# B&R Automation Studio project Teknologia25 (part 10)

#### rotationProgram.st
```iecst
ACTION rotationTask:
	positionContainerRotation[0].initXPos := 0.180;
	positionContainerRotation[0].initYPos := 0.060;
	positionContainerRotation[1].initXPos := 0.060;
	positionContainerRotation[1].initYPos := 0.060;
	positionContainerRotation[2].initXPos := 0.060;
	positionContainerRotation[2].initYPos := 0.180;
	positionContainerRotation[3].initXPos := 0.180;
	positionContainerRotation[3].initYPos := 0.180;

	gWorkStations[0].par.xLocation										:= 0.180;
	gWorkStations[0].par.yLocation										:= 0.060;
	gWorkStations[0].par.nextStationSelector							:= '1';
	gWorkStations[0].par.processTime									:= 0;
	gWorkStations[0].par.pathRouting									:= 1;
	gWorkStations[0].par.landBeforeProcess								:= FALSE;
	gWorkStations[0].par.ArcMovement									:= FALSE;

	gWorkStations[1].par.xLocation										:= 0.060;
	gWorkStations[1].par.yLocation										:= 0.180;
	gWorkStations[1].par.nextStationSelector							:= '0';
	gWorkStations[1].par.processTime									:= WorkStation2And3MovementTimer;
	gWorkStations[1].par.pathRouting									:= 2;
	gWorkStations[1].par.landBeforeProcess								:= TRUE;
	gWorkStations[1].par.ArcMovement									:= FALSE;

	CASE em.substate OF
		14000:
			em.description := 'Move shuttle to pre pos';
			tempShuttleCounter := 0;
			MC_BR_MoveInPlaneAsync_Acp6D_0.Parameters.Acceleration := gAcp6DCtrl.Par.Acceleration;
			MC_BR_MoveInPlaneAsync_Acp6D_0.Parameters.Velocity := gAcp6DCtrl.Par.Velocity;
			FOR i := 0 TO UINT_TO_USINT(localCurrentNumShuttles-1) DO
				MC_BR_MoveInPlaneAsync_Acp6D_0.Parameters.AsyncPar[i].Shuttle := ADR(gAcp6DCtrl.Status.ShuttleInfo[i].shuttleRef);
				MC_BR_MoveInPlaneAsync_Acp6D_0.Parameters.AsyncPar[i].X := positionContainerRotation[i].initXPos;
				MC_BR_MoveInPlaneAsync_Acp6D_0.Parameters.AsyncPar[i].Y := positionContainerRotation[i].initYPos;
			END_FOR
			MC_BR_MoveInPlaneAsync_Acp6D_0.Execute := TRUE;
			IF MC_BR_MoveInPlaneAsync_Acp6D_0.Acknowledge THEN
				MC_BR_MoveInPlaneAsync_Acp6D_0.Execute := FALSE;
				em.substate := 14010;
			END_IF

		14010:
			em.description := 'Move shuttle 2 towards workstation 0';
			MC_BR_MoveInPlane_Acp6D_0.Parameters.Acceleration := gAcp6DCtrl.Par.Acceleration;
			MC_BR_MoveInPlane_Acp6D_0.Parameters.Velocity := gAcp6DCtrl.Par.Velocity;
			MC_BR_MoveInPlane_Acp6D_0.Shuttle := ADR(gAcp6DCtrl.Status.ShuttleInfo[1].shuttleRef);;
			MC_BR_MoveInPlane_Acp6D_0.Parameters.Position.X := gWorkStations[0].par.xLocation;;
			MC_BR_MoveInPlane_Acp6D_0.Parameters.Position.Y := gWorkStations[0].par.yLocation;
			MC_BR_MoveInPlane_Acp6D_0.Parameters.Path := 0; //direct
			MC_BR_MoveInPlane_Acp6D_0.Parameters.Mode := 0;
			MC_BR_MoveInPlane_Acp6D_0.Execute := TRUE;
			IF MC_BR_MoveInPlane_Acp6D_0.Acknowledge THEN
				MC_BR_MoveInPlane_Acp6D_0.Execute := FALSE;
				em.substate := 14020;
			END_IF

		14020:
			em.description := 'Move shuttle 3 towards workstation 0';
			MC_BR_MoveInPlane_Acp6D_0.Parameters.Acceleration := gAcp6DCtrl.Par.Acceleration;
			MC_BR_MoveInPlane_Acp6D_0.Parameters.Velocity := gAcp6DCtrl.Par.Velocity;
			MC_BR_MoveInPlane_Acp6D_0.Shuttle := ADR(gAcp6DCtrl.Status.ShuttleInfo[2].shuttleRef);;
			MC_BR_MoveInPlane_Acp6D_0.Parameters.Position.X := gWorkStations[0].par.xLocation;;
			MC_BR_MoveInPlane_Acp6D_0.Parameters.Position.Y := gWorkStations[0].par.yLocation;
			MC_BR_MoveInPlane_Acp6D_0.Parameters.Path := 2; //Y then X
			MC_BR_MoveInPlane_Acp6D_0.Parameters.Mode := 0;
			MC_BR_MoveInPlane_Acp6D_0.Execute := TRUE;
			IF MC_BR_MoveInPlane_Acp6D_0.Acknowledge THEN
				MC_BR_MoveInPlane_Acp6D_0.Execute := FALSE;
				em.substate := 14030;
			END_IF

		14030:
			em.description := 'Move shuttle 4 towards workstation 1';
			MC_BR_MoveInPlane_Acp6D_0.Parameters.Acceleration := gAcp6DCtrl.Par.Acceleration;
			MC_BR_MoveInPlane_Acp6D_0.Parameters.Velocity := gAcp6DCtrl.Par.Velocity;
			MC_BR_MoveInPlane_Acp6D_0.Shuttle := ADR(gAcp6DCtrl.Status.ShuttleInfo[3].shuttleRef);;
			MC_BR_MoveInPlane_Acp6D_0.Parameters.Position.X := 0.060;
			MC_BR_MoveInPlane_Acp6D_0.Parameters.Position.Y := 0.180;
			MC_BR_MoveInPlane_Acp6D_0.Parameters.Path := 0; //direct
			MC_BR_MoveInPlane_Acp6D_0.Parameters.Mode := 0;
			MC_BR_MoveInPlane_Acp6D_0.Execute := TRUE;
			IF MC_BR_MoveInPlane_Acp6D_0.Acknowledge THEN
				MC_BR_MoveInPlane_Acp6D_0.Execute := FALSE;
				em.substate := 14040;
			END_IF

		14040:
			em.description := 'Move shuttle 4 towards workstation 1';
			MC_BR_MoveInPlane_Acp6D_0.Parameters.Acceleration := gAcp6DCtrl.Par.Acceleration;
			MC_BR_MoveInPlane_Acp6D_0.Parameters.Velocity := gAcp6DCtrl.Par.Velocity;
			MC_BR_MoveInPlane_Acp6D_0.Shuttle := ADR(gAcp6DCtrl.Status.ShuttleInfo[3].shuttleRef);;
			MC_BR_MoveInPlane_Acp6D_0.Parameters.Position.X := gWorkStations[0].par.xLocation;
			MC_BR_MoveInPlane_Acp6D_0.Parameters.Position.Y := gWorkStations[0].par.yLocation;
			MC_BR_MoveInPlane_Acp6D_0.Parameters.Path := 2; //direct
			MC_BR_MoveInPlane_Acp6D_0.Parameters.Mode := 0;
			MC_BR_MoveInPlane_Acp6D_0.Execute := TRUE;
			IF MC_BR_MoveInPlane_Acp6D_0.Acknowledge THEN
				MC_BR_MoveInPlane_Acp6D_0.Execute := FALSE;
				em.substate := 14050;
			END_IF
	END_CASE

END_ACTION

ACTION rotationStation:
	CASE cm.state OF
		// Display station at image
		//'<foreignObject x="20" y="20" width="300" height="300"><img src="Media/statusGreen.png" height="300" width="300"/>'
		//brsstrcat(ADR(showWorkStations),ADR('<foreingObject x="'));
		//brdkStrCat(ADR(showWorkStations), ADR(testDraw));
		//brdkStrCat(ADR(showWorkStations),'<foreingObject x="');

		0:
			//Check what shuttle is on top of workstation
			FOR k := 0 TO NUM_SHUTTLES DO
				IF((gAcp6DCtrl.Status.ShuttleInfo[k].Position.X > pWorkStations.par.xLocation - MARGIN AND gAcp6DCtrl.Status.ShuttleInfo[k].Position.X < pWorkStations.par.xLocation + MARGIN) AND
					gAcp6DCtrl.Status.ShuttleInfo[k].Position.Y > pWorkStations.par.yLocation - MARGIN AND gAcp6DCtrl.Status.ShuttleInfo[k].Position.Y < pWorkStations.par.yLocation + MARGIN) THEN
					IF gAcp6DCtrl.Status.ShuttleInfo[k].State = mcACP6D_SH_STATE_IDLING THEN
						pWorkStations.par.tempShuttleID := k;
						cm.state := 10;
					END_IF
				END_IF
			END_FOR

		10:
			//Move first workstation
			pWorkStations.MC_BR_MoveInPlane_Acp6D_0.Shuttle := ADR(gAcp6DCtrl.Status.ShuttleInfo[pWorkStations.par.tempShuttleID].shuttleRef);
			pWorkStations.MC_BR_MoveInPlane_Acp6D_0.Parameters.Velocity := gAcp6DCtrl.Par.Velocity;
			pWorkStations.MC_BR_MoveInPlane_Acp6D_0.Parameters.Acceleration := gAcp6DCtrl.Par.Acceleration;
			pWorkStations.MC_BR_MoveInPlane_Acp6D_0.Parameters.Position.X := 0.360;
			pWorkStations.MC_BR_MoveInPlane_Acp6D_0.Parameters.Position.Y := 0.120;
			pWorkStations.MC_BR_MoveInPlane_Acp6D_0.Parameters.Mode := 0; //Absolute
			pWorkStations.MC_BR_MoveInPlane_Acp6D_0.Parameters.Path := 1; //0 Diagonal, 1 First X then Y, 2 First Y then X
			pWorkStations.MC_BR_MoveInPlane_Acp6D_0.Execute := TRUE;
			IF pWorkStations.MC_BR_MoveInPlane_Acp6D_0.Done THEN
				pWorkStations.MC_BR_MoveInPlane_Acp6D_0.Execute := FALSE;
				cm.state := 20;
			END_IF

		20:
			//Rotate 90 degress
			em.cmd.sc := FALSE;
			pWorkStations.MC_BR_RotaryMotion_Acp6D_0.Shuttle := ADR(gAcp6DCtrl.Status.ShuttleInfo[pWorkStations.par.tempShuttleID].shuttleRef);
			pWorkStations.MC_BR_RotaryMotion_Acp6D_0.Parameters.Acceleration := gAcp6DCtrl.Par.rotationAcceleration;
			pWorkStations.MC_BR_RotaryMotion_Acp6D_0.Parameters.Velocity := gAcp6DCtrl.Par.rotationVelocity;
			pWorkStations.MC_BR_RotaryMotion_Acp6D_0.Parameters.Angle := 1.57079633; //90 degress
			pWorkStations.MC_BR_RotaryMotion_Acp6D_0.Parameters.Mode := 0;
			pWorkStations.MC_BR_RotaryMotion_Acp6D_0.Execute := TRUE;
			IF pWorkStations.MC_BR_RotaryMotion_Acp6D_0.Done THEN
				pWorkStations.MC_BR_RotaryMotion_Acp6D_0.Execute := FALSE;
				cm.state := 30;
			END_IF

		30:
			//Move
			//em.cmd.sc := FALSE;
			pWorkStations.MC_BR_MoveInPlane_Acp6D_0.Shuttle := ADR(gAcp6DCtrl.Status.ShuttleInfo[pWorkStations.par.tempShuttleID].shuttleRef);
			pWorkStations.MC_BR_MoveInPlane_Acp6D_0.Parameters.Velocity := gAcp6DCtrl.Par.Velocity;
			pWorkStations.MC_BR_MoveInPlane_Acp6D_0.Parameters.Acceleration := gAcp6DCtrl.Par.Acceleration;
			pWorkStations.MC_BR_MoveInPlane_Acp6D_0.Parameters.Position.X := 0.420;
			pWorkStations.MC_BR_MoveInPlane_Acp6D_0.Parameters.Position.Y := 0.120;
			pWorkStations.MC_BR_MoveInPlane_Acp6D_0.Parameters.Mode := 0; //Absolute
			pWorkStations.MC_BR_MoveInPlane_Acp6D_0.Parameters.Path := 1; //0 Diagonal, 1 First X then Y, 2 First Y then X
			pWorkStations.MC_BR_MoveInPlane_Acp6D_0.Execute := TRUE;
			IF pWorkStations.MC_BR_MoveInPlane_Acp6D_0.Acknowledge THEN
				pWorkStations.MC_BR_MoveInPlane_Acp6D_0.Execute := FALSE;
				cm.state := 40;
			END_IF

		40:
			//em.cmd.sc := FALSE;
			pWorkStations.TON_0.IN := TRUE;
			pWorkStations.TON_0.PT := t#100ms;
			IF pWorkStations.TON_0.Q THEN
				pWorkStations.TON_0.IN := FALSE;
				cm.state := 50;
			END_IF

		50:
			//Move
			//em.cmd.sc := FALSE;
			pWorkStations.MC_BR_MoveInPlane_Acp6D_0.Shuttle := ADR(gAcp6DCtrl.Status.ShuttleInfo[pWorkStations.par.tempShuttleID].shuttleRef);
			pWorkStations.MC_BR_MoveInPlane_Acp6D_0.Parameters.Velocity := gAcp6DCtrl.Par.Velocity;
			pWorkStations.MC_BR_MoveInPlane_Acp6D_0.Parameters.Acceleration := gAcp6DCtrl.Par.Acceleration;
			pWorkStations.MC_BR_MoveInPlane_Acp6D_0.Parameters.Position.X := 0.360;
			pWorkStations.MC_BR_MoveInPlane_Acp6D_0.Parameters.Position.Y := 0.120;
			pWorkStations.MC_BR_MoveInPlane_Acp6D_0.Parameters.Mode := 0; //Absolute
			pWorkStations.MC_BR_MoveInPlane_Acp6D_0.Parameters.Path := 1; //0 Diagonal, 1 First X then Y, 2 First Y then X
			pWorkStations.MC_BR_MoveInPlane_Acp6D_0.Execute := TRUE;
			IF pWorkStations.MC_BR_MoveInPlane_Acp6D_0.Acknowledge THEN
				pWorkStations.MC_BR_MoveInPlane_Acp6D_0.Execute := FALSE;
				cm.state := 60;
			END_IF

		60:
			//Rotate 90 degress
			em.cmd.sc := FALSE;
			pWorkStations.MC_BR_RotaryMotion_Acp6D_0.Shuttle := ADR(gAcp6DCtrl.Status.ShuttleInfo[pWorkStations.par.tempShuttleID].shuttleRef);
			pWorkStations.MC_BR_RotaryMotion_Acp6D_0.Parameters.Acceleration := gAcp6DCtrl.Par.rotationAcceleration;
			pWorkStations.MC_BR_RotaryMotion_Acp6D_0.Parameters.Velocity := gAcp6DCtrl.Par.rotationVelocity;
			pWorkStations.MC_BR_RotaryMotion_Acp6D_0.Parameters.Angle := 3.14159265; //180 degress
			pWorkStations.MC_BR_RotaryMotion_Acp6D_0.Parameters.Mode := 0;
			pWorkStations.MC_BR_RotaryMotion_Acp6D_0.Execute := TRUE;
			IF pWorkStations.MC_BR_RotaryMotion_Acp6D_0.Done THEN
				pWorkStations.MC_BR_RotaryMotion_Acp6D_0.Execute := FALSE;
				cm.state := 70;
			END_IF

		70:
			//Move
			//em.cmd.sc := FALSE;
			pWorkStations.MC_BR_MoveInPlane_Acp6D_0.Shuttle := ADR(gAcp6DCtrl.Status.ShuttleInfo[pWorkStations.par.tempShuttleID].shuttleRef);
			pWorkStations.MC_BR_MoveInPlane_Acp6D_0.Parameters.Velocity := gAcp6DCtrl.Par.Velocity;
			pWorkStations.MC_BR_MoveInPlane_Acp6D_0.Parameters.Acceleration := gAcp6DCtrl.Par.Acceleration;
			pWorkStations.MC_BR_MoveInPlane_Acp6D_0.Parameters.Position.X := 0.420;
			pWorkStations.MC_BR_MoveInPlane_Acp6D_0.Parameters.Position.Y := 0.120;
			pWorkStations.MC_BR_MoveInPlane_Acp6D_0.Parameters.Mode := 0; //Absolute
			pWorkStations.MC_BR_MoveInPlane_Acp6D_0.Parameters.Path := 1; //0 Diagonal, 1 First X then Y, 2 First Y then X
			pWorkStations.MC_BR_MoveInPlane_Acp6D_0.Execute := TRUE;
			IF pWorkStations.MC_BR_MoveInPlane_Acp6D_0.Acknowledge THEN
				pWorkStations.MC_BR_MoveInPlane_Acp6D_0.Execute := FALSE;
				cm.state := 80;
			END_IF

		80:
			//em.cmd.sc := FALSE;
			pWorkStations.TON_0.IN := TRUE;
			pWorkStations.TON_0.PT := t#100ms;
			IF pWorkStations.TON_0.Q THEN
				pWorkStations.TON_0.IN := FALSE;
				cm.state := 90;
			END_IF

		90:
			//Move
			//em.cmd.sc := FALSE;
			pWorkStations.MC_BR_MoveInPlane_Acp6D_0.Shuttle := ADR(gAcp6DCtrl.Status.ShuttleInfo[pWorkStations.par.tempShuttleID].shuttleRef);
			pWorkStations.MC_BR_MoveInPlane_Acp6D_0.Parameters.Velocity := gAcp6DCtrl.Par.Velocity;
			pWorkStations.MC_BR_MoveInPlane_Acp6D_0.Parameters.Acceleration := gAcp6DCtrl.Par.Acceleration;
			pWorkStations.MC_BR_MoveInPlane_Acp6D_0.Parameters.Position.X := 0.360;
			pWorkStations.MC_BR_MoveInPlane_Acp6D_0.Parameters.Position.Y := 0.120;
			pWorkStations.MC_BR_MoveInPlane_Acp6D_0.Parameters.Mode := 0; //Absolute
			pWorkStations.MC_BR_MoveInPlane_Acp6D_0.Parameters.Path := 1; //0 Diagonal, 1 First X then Y, 2 First Y then X
			pWorkStations.MC_BR_MoveInPlane_Acp6D_0.Execute := TRUE;
			IF pWorkStations.MC_BR_MoveInPlane_Acp6D_0.Acknowledge THEN
				pWorkStations.MC_BR_MoveInPlane_Acp6D_0.Execute := FALSE;
				cm.state := 100;
			END_IF

		100:
			//Rotate 90 degress
			em.cmd.sc := FALSE;
			pWorkStations.MC_BR_RotaryMotion_Acp6D_0.Shuttle := ADR(gAcp6DCtrl.Status.ShuttleInfo[pWorkStations.par.tempShuttleID].shuttleRef);
			pWorkStations.MC_BR_RotaryMotion_Acp6D_0.Parameters.Acceleration := gAcp6DCtrl.Par.rotationAcceleration;
			pWorkStations.MC_BR_RotaryMotion_Acp6D_0.Parameters.Velocity := gAcp6DCtrl.Par.rotationVelocity;
			pWorkStations.MC_BR_RotaryMotion_Acp6D_0.Parameters.Angle := 4.71238898; //270 degress
			pWorkStations.MC_BR_RotaryMotion_Acp6D_0.Parameters.Mode := 0;
			pWorkStations.MC_BR_RotaryMotion_Acp6D_0.Execute := TRUE;
			IF pWorkStations.MC_BR_RotaryMotion_Acp6D_0.Done THEN
				pWorkStations.MC_BR_RotaryMotion_Acp6D_0.Execute := FALSE;
				cm.state := 110;
			END_IF

		110:
			//Move
			//em.cmd.sc := FALSE;
			pWorkStations.MC_BR_MoveInPlane_Acp6D_0.Shuttle := ADR(gAcp6DCtrl.Status.ShuttleInfo[pWorkStations.par.tempShuttleID].shuttleRef);
			pWorkStations.MC_BR_MoveInPlane_Acp6D_0.Parameters.Velocity := gAcp6DCtrl.Par.Velocity;
			pWorkStations.MC_BR_MoveInPlane_Acp6D_0.Parameters.Acceleration := gAcp6DCtrl.Par.Acceleration;
			pWorkStations.MC_BR_MoveInPlane_Acp6D_0.Parameters.Position.X := 0.420;
			pWorkStations.MC_BR_MoveInPlane_Acp6D_0.Parameters.Position.Y := 0.120;
			pWorkStations.MC_BR_MoveInPlane_Acp6D_0.Parameters.Mode := 0; //Absolute
			pWorkStations.MC_BR_MoveInPlane_Acp6D_0.Parameters.Path := 1; //0 Diagonal, 1 First X then Y, 2 First Y then X
			pWorkStations.MC_BR_MoveInPlane_Acp6D_0.Execute := TRUE;
			IF pWorkStations.MC_BR_MoveInPlane_Acp6D_0.Acknowledge THEN
				pWorkStations.MC_BR_MoveInPlane_Acp6D_0.Execute := FALSE;
				cm.state := 120;
			END_IF

		120:
			//em.cmd.sc := FALSE;
			pWorkStations.TON_0.IN := TRUE;
			pWorkStations.TON_0.PT := t#100ms;
			IF pWorkStations.TON_0.Q THEN
				pWorkStations.TON_0.IN := FALSE;
				cm.state := 130;
			END_IF

		130:
			//Move
			//em.cmd.sc := FALSE;
			pWorkStations.MC_BR_MoveInPlane_Acp6D_0.Shuttle := ADR(gAcp6DCtrl.Status.ShuttleInfo[pWorkStations.par.tempShuttleID].shuttleRef);
			pWorkStations.MC_BR_MoveInPlane_Acp6D_0.Parameters.Velocity := gAcp6DCtrl.Par.Velocity;
			pWorkStations.MC_BR_MoveInPlane_Acp6D_0.Parameters.Acceleration := gAcp6DCtrl.Par.Acceleration;
			pWorkStations.MC_BR_MoveInPlane_Acp6D_0.Parameters.Position.X := 0.360;
			pWorkStations.MC_BR_MoveInPlane_Acp6D_0.Parameters.Position.Y := 0.120;
			pWorkStations.MC_BR_MoveInPlane_Acp6D_0.Parameters.Mode := 0; //Absolute
			pWorkStations.MC_BR_MoveInPlane_Acp6D_0.Parameters.Path := 1; //0 Diagonal, 1 First X then Y, 2 First Y then X
			pWorkStations.MC_BR_MoveInPlane_Acp6D_0.Execute := TRUE;
			IF pWorkStations.MC_BR_MoveInPlane_Acp6D_0.Acknowledge THEN
				pWorkStations.MC_BR_MoveInPlane_Acp6D_0.Execute := FALSE;
				cm.state := 140;
			END_IF

		140:
			//Rotate
			em.cmd.sc := FALSE;
			pWorkStations.MC_BR_RotaryMotion_Acp6D_0.Shuttle := ADR(gAcp6DCtrl.Status.ShuttleInfo[pWorkStations.par.tempShuttleID].shuttleRef);
			pWorkStations.MC_BR_RotaryMotion_Acp6D_0.Parameters.Acceleration := gAcp6DCtrl.Par.rotationAcceleration;
			pWorkStations.MC_BR_RotaryMotion_Acp6D_0.Parameters.Velocity := gAcp6DCtrl.Par.rotationVelocity; //RPM
			pWorkStations.MC_BR_RotaryMotion_Acp6D_0.Parameters.Angle := 0; //0 degress
			pWorkStations.MC_BR_RotaryMotion_Acp6D_0.Parameters.Mode := 1;
			pWorkStations.MC_BR_RotaryMotion_Acp6D_0.Execute := TRUE;
			IF pWorkStations.MC_BR_RotaryMotion_Acp6D_0.Done THEN
				pWorkStations.MC_BR_RotaryMotion_Acp6D_0.Execute := FALSE;
				cm.state := 145;
			END_IF

		145:
			em.cmd.sc := FALSE;
			pWorkStations.MC_BR_RotaryMotionSpin_Acp6D_0.Shuttle := ADR(gAcp6DCtrl.Status.ShuttleInfo[pWorkStations.par.tempShuttleID].shuttleRef);
			pWorkStations.MC_BR_RotaryMotionSpin_Acp6D_0.Parameters.Velocity := gAcp6DCtrl.Par.rotationVelocity;
			pWorkStations.MC_BR_RotaryMotionSpin_Acp6D_0.Parameters.Acceleration := gAcp6DCtrl.Par.rotationAcceleration;
			pWorkStations.MC_BR_RotaryMotionSpin_Acp6D_0.Parameters.Duration := 5;
			pWorkStations.MC_BR_RotaryMotionSpin_Acp6D_0.Execute := TRUE;
			IF pWorkStations.MC_BR_RotaryMotionSpin_Acp6D_0.Done THEN
				pWorkStations.MC_BR_RotaryMotionSpin_Acp6D_0.Execute := FALSE;
				cm.state := 150;
			END_IF

		150:
			//Move
			pWorkStations.MC_BR_MoveInPlane_Acp6D_0.Shuttle := ADR(gAcp6DCtrl.Status.ShuttleInfo[pWorkStations.par.tempShuttleID].shuttleRef);
			pWorkStations.MC_BR_MoveInPlane_Acp6D_0.Parameters.Velocity := gAcp6DCtrl.Par.Velocity;
			pWorkStations.MC_BR_MoveInPlane_Acp6D_0.Parameters.Acceleration := gAcp6DCtrl.Par.Acceleration;
			pWorkStations.MC_BR_MoveInPlane_Acp6D_0.Parameters.Position.X := 0.060;
			pWorkStations.MC_BR_MoveInPlane_Acp6D_0.Parameters.Position.Y := 0.180;
			pWorkStations.MC_BR_MoveInPlane_Acp6D_0.Parameters.Mode := 0; //Absolute
			pWorkStations.MC_BR_MoveInPlane_Acp6D_0.Parameters.Path := 2; //0 Diagonal, 1 First X then Y, 2 First Y then X
			pWorkStations.MC_BR_MoveInPlane_Acp6D_0.Execute := TRUE;
			IF pWorkStations.MC_BR_MoveInPlane_Acp6D_0.Acknowledge THEN
				pWorkStations.MC_BR_MoveInPlane_Acp6D_0.Execute := FALSE;
				cm.state := 160;
			END_IF

		160:
			//Move
			pWorkStations.MC_BR_MoveInPlane_Acp6D_0.Shuttle := ADR(gAcp6DCtrl.Status.ShuttleInfo[pWorkStations.par.tempShuttleID].shuttleRef);
			pWorkStations.MC_BR_MoveInPlane_Acp6D_0.Parameters.Velocity := gAcp6DCtrl.Par.Velocity;
			pWorkStations.MC_BR_MoveInPlane_Acp6D_0.Parameters.Acceleration := gAcp6DCtrl.Par.Acceleration;
			pWorkStations.MC_BR_MoveInPlane_Acp6D_0.Parameters.Position.X := gWorkStations[0].par.xLocation;
			pWorkStations.MC_BR_MoveInPlane_Acp6D_0.Parameters.Position.Y := gWorkStations[0].par.yLocation;
			pWorkStations.MC_BR_MoveInPlane_Acp6D_0.Parameters.Mode := 0; //Absolute
			pWorkStations.MC_BR_MoveInPlane_Acp6D_0.Parameters.Path := 2; //0 Diagonal, 1 First X then Y, 2 First Y then X
			pWorkStations.MC_BR_MoveInPlane_Acp6D_0.Execute := TRUE;
			IF pWorkStations.MC_BR_MoveInPlane_Acp6D_0.Acknowledge THEN
				pWorkStations.MC_BR_MoveInPlane_Acp6D_0.Execute := FALSE;
				cm.state := 0;
			END_IF

	END_CASE

	//Calls
	pWorkStations.MC_BR_MoveInPlane_Acp6D_0();
	pWorkStations.MC_BR_MoveArc_Acp6D_0();
	pWorkStations.MC_BR_ShLevitation_Acp6D_0();
	pWorkStations.MC_BR_RotaryMotion_Acp6D_0();
	pWorkStations.MC_BR_RotaryMotionSpin_Acp6D_0();
	pWorkStations.TON_0();
	cm();

END_ACTION
```

#### steelSheet.st
```iecst
ACTION steelSheetTask:
	positionContainerSteelSheet[0].initXPos := 0.060;
	positionContainerSteelSheet[0].initYPos := 0.060;
	positionContainerSteelSheet[1].initXPos := 0.180;
	positionContainerSteelSheet[1].initYPos := 0.060;
	positionContainerSteelSheet[2].initXPos := 0.300;
	positionContainerSteelSheet[2].initYPos := 0.060;
	positionContainerSteelSheet[3].initXPos := 0.420;
	positionContainerSteelSheet[3].initYPos := 0.060;

	gWorkStations[0].par.xLocation										:= 0.060;
	gWorkStations[0].par.yLocation										:= 0.060;
	gWorkStations[0].par.nextStationSelector							:= '0';
	gWorkStations[0].par.processTime									:= 0;
	gWorkStations[0].par.pathRouting									:= 0;
	gWorkStations[0].par.landBeforeProcess								:= FALSE;
	gWorkStations[0].par.ArcMovement									:= FALSE;

	gWorkStations[1].par.xLocation										:= 0.180;
	gWorkStations[1].par.yLocation										:= 0.060;
	gWorkStations[1].par.nextStationSelector							:= '1';
	gWorkStations[1].par.processTime									:= 0;
	gWorkStations[1].par.pathRouting									:= 0;
	gWorkStations[1].par.landBeforeProcess								:= FALSE;
	gWorkStations[1].par.ArcMovement									:= FALSE;

	gWorkStations[2].par.xLocation										:= 0.300;
	gWorkStations[2].par.yLocation										:= 0.060;
	gWorkStations[2].par.nextStationSelector							:= '2';
	gWorkStations[2].par.processTime									:= 0;
	gWorkStations[2].par.pathRouting									:= 0;
	gWorkStations[2].par.landBeforeProcess								:= FALSE;
	gWorkStations[2].par.ArcMovement									:= FALSE;

	gWorkStations[3].par.xLocation										:= 0.420;
	gWorkStations[3].par.yLocation										:= 0.060;
	gWorkStations[3].par.nextStationSelector							:= '3';
	gWorkStations[3].par.processTime									:= 0;
	gWorkStations[3].par.pathRouting									:= 0;
	gWorkStations[3].par.landBeforeProcess								:= FALSE;
	gWorkStations[3].par.ArcMovement									:= FALSE;

	// Make sure all shuttles have finish movement
	sheetMoveDone := TRUE;
//	FOR i := 0 TO NR_OF_WORKSTATIONS DO
//		IF NOT gWorkStations[i].MC_BR_Move6D_Acp6D_0.Done THEN
//			sheetMoveDone := FALSE;
//		END_IF
//	END_FOR
	FOR i := 0 TO NR_OF_WORKSTATIONS DO
		IF NOT gWorkStations[i].MC_BR_MoveInPlane_Acp6D_0.Done THEN
			sheetMoveDone := FALSE;
		END_IF
	END_FOR

	CASE em.substate OF
		15000:
			em.description := 'Move shuttle to pre pos';
			tempShuttleCounter := 0;
			MC_BR_MoveInPlaneAsync_Acp6D_0.Parameters.Acceleration := gAcp6DCtrl.Par.Acceleration;
			MC_BR_MoveInPlaneAsync_Acp6D_0.Parameters.Velocity := gAcp6DCtrl.Par.Velocity;
			FOR i := 0 TO UINT_TO_USINT(localCurrentNumShuttles-1) DO
				MC_BR_MoveInPlaneAsync_Acp6D_0.Parameters.AsyncPar[i].Shuttle := ADR(gAcp6DCtrl.Status.ShuttleInfo[i].shuttleRef);
				MC_BR_MoveInPlaneAsync_Acp6D_0.Parameters.AsyncPar[i].X := positionContainerSteelSheet[i].initXPos;
				MC_BR_MoveInPlaneAsync_Acp6D_0.Parameters.AsyncPar[i].Y := positionContainerSteelSheet[i].initYPos;
				MC_BR_MoveInPlaneAsync_Acp6D_0.Parameters.AsyncPar[i].Y := positionContainerSteelSheet[i].initYPos;
			END_FOR
			MC_BR_MoveInPlaneAsync_Acp6D_0.Execute := TRUE;
			IF MC_BR_MoveInPlaneAsync_Acp6D_0.Acknowledge THEN
				MC_BR_MoveInPlaneAsync_Acp6D_0.Execute := FALSE;
				em.substate := 15010;
			END_IF

		15010:
			em.description := 'Shuttle moves at a higher levitation hight';

	END_CASE

END_ACTION

ACTION steelSheetStation:
	CASE cm.state OF
		0:
			//Check what shuttle is on top of workstation
			FOR k := 0 TO NUM_SHUTTLES DO
				IF((gAcp6DCtrl.Status.ShuttleInfo[k].Position.X > pWorkStations.par.xLocation - MARGIN AND gAcp6DCtrl.Status.ShuttleInfo[k].Position.X < pWorkStations.par.xLocation + MARGIN) AND
					gAcp6DCtrl.Status.ShuttleInfo[k].Position.Y > pWorkStations.par.yLocation - MARGIN AND gAcp6DCtrl.Status.ShuttleInfo[k].Position.Y < pWorkStations.par.yLocation + MARGIN) THEN
					IF gAcp6DCtrl.Status.ShuttleInfo[k].State = mcACP6D_SH_STATE_IDLING THEN
						pWorkStations.par.tempShuttleID := k;
						cm.state := 5;
					END_IF
				END_IF
			END_FOR

		5:
			// Levitate to sheet flying height
			pWorkStations.MC_BR_MoveShortAxis_Acp6D_0.Shuttle := ADR(gAcp6DCtrl.Status.ShuttleInfo[pWorkStations.par.tempShuttleID].shuttleRef);
			pWorkStations.MC_BR_MoveShortAxis_Acp6D_0.Parameters.Position.Z := steelSheetFlyingHeight;
			pWorkStations.MC_BR_MoveShortAxis_Acp6D_0.Parameters.Position.Rx := 0;
			pWorkStations.MC_BR_MoveShortAxis_Acp6D_0.Parameters.Position.Ry := 0;
			pWorkStations.MC_BR_MoveShortAxis_Acp6D_0.Parameters.Position.Rz := 0;
			pWorkStations.MC_BR_MoveShortAxis_Acp6D_0.Parameters.Velocity.Z := 0.01;
			pWorkStations.MC_BR_MoveShortAxis_Acp6D_0.Execute := TRUE;
			IF pWorkStations.MC_BR_MoveShortAxis_Acp6D_0.Done THEN
				pWorkStations.MC_BR_MoveShortAxis_Acp6D_0.Execute := FALSE;
				cm.state := 10;
			END_IF

		10:
//			pWorkStations.MC_BR_Move6D_Acp6D_0.Shuttle := ADR(gAcp6DCtrl.Status.ShuttleInfo[pWorkStations.par.tempShuttleID].shuttleRef);
//			pWorkStations.MC_BR_Move6D_Acp6D_0.Parameters.InPlane.Velocity := stainlessVelocity;
//			pWorkStations.MC_BR_Move6D_Acp6D_0.Parameters.InPlane.Acceleration := stainlessAcceleration;
//			pWorkStations.MC_BR_Move6D_Acp6D_0.Parameters.InPlane.Position.X := pWorkStations.par.xLocation;
//			pWorkStations.MC_BR_Move6D_Acp6D_0.Parameters.InPlane.Position.Y := 0.180;
//			pWorkStations.MC_BR_Move6D_Acp6D_0.Parameters.ShortAxis.Position.Z := steelSheetFlyingHeight;
//			pWorkStations.MC_BR_Move6D_Acp6D_0.Parameters.ShortAxis.Position.Rx := 0;
//			pWorkStations.MC_BR_Move6D_Acp6D_0.Parameters.ShortAxis.Position.Ry := 0;
//			pWorkStations.MC_BR_Move6D_Acp6D_0.Parameters.ShortAxis.Position.Rz := 0;
//			pWorkStations.MC_BR_Move6D_Acp6D_0.Execute := TRUE;
//			IF pWorkStations.MC_BR_Move6D_Acp6D_0.Done AND sheetMoveDone THEN
//				pWorkStations.MC_BR_Move6D_Acp6D_0.Execute := FALSE;
//				cm.state := 30;
//			END_IF

			pWorkStations.MC_BR_MoveInPlane_Acp6D_0.Shuttle := ADR(gAcp6DCtrl.Status.ShuttleInfo[pWorkStations.par.tempShuttleID].shuttleRef);
			pWorkStations.MC_BR_MoveInPlane_Acp6D_0.Parameters.Velocity := stainlessVelocity;
			pWorkStations.MC_BR_MoveInPlane_Acp6D_0.Parameters.Acceleration := stainlessAcceleration;
			pWorkStations.MC_BR_MoveInPlane_Acp6D_0.Parameters.Position.X := pWorkStations.par.xLocation;
			pWorkStations.MC_BR_MoveInPlane_Acp6D_0.Parameters.Position.Y := 0.180;

			pWorkStations.MC_BR_MoveInPlane_Acp6D_0.Execute := TRUE;
			IF pWorkStations.MC_BR_MoveInPlane_Acp6D_0.Done AND sheetMoveDone THEN
				pWorkStations.MC_BR_MoveInPlane_Acp6D_0.Execute := FALSE;
				cm.state := 15;
			END_IF

		15:
			pWorkStations.TON_0.IN := TRUE;
			pWorkStations.TON_0.PT := stainlessWaitTime;
			IF pWorkStations.TON_0.Q THEN
				pWorkStations.TON_0.IN := FALSE;
				cm.state := 30;
			END_IF

		30:
//			pWorkStations.MC_BR_Move6D_Acp6D_0.Shuttle := ADR(gAcp6DCtrl.Status.ShuttleInfo[pWorkStations.par.tempShuttleID].shuttleRef);
//			pWorkStations.MC_BR_Move6D_Acp6D_0.Parameters.InPlane.Velocity := stainlessVelocity;
//			pWorkStations.MC_BR_Move6D_Acp6D_0.Parameters.InPlane.Acceleration := stainlessAcceleration;
//			pWorkStations.MC_BR_Move6D_Acp6D_0.Parameters.InPlane.Position.X := pWorkStations.par.xLocation;
//			pWorkStations.MC_BR_Move6D_Acp6D_0.Parameters.InPlane.Position.Y := 0.060;
//			pWorkStations.MC_BR_Move6D_Acp6D_0.Parameters.ShortAxis.Position.Rx := 0;
//			pWorkStations.MC_BR_Move6D_Acp6D_0.Parameters.ShortAxis.Position.Ry := 0;
//			pWorkStations.MC_BR_Move6D_Acp6D_0.Parameters.ShortAxis.Position.Rz := 0;
//			pWorkStations.MC_BR_Move6D_Acp6D_0.Parameters.ShortAxis.Position.Z := steelSheetFlyingHeight;
//			pWorkStations.MC_BR_Move6D_Acp6D_0.Execute := TRUE;
//			IF pWorkStations.MC_BR_Move6D_Acp6D_0.Done AND sheetMoveDone THEN
//				pWorkStations.MC_BR_Move6D_Acp6D_0.Execute := FALSE;
//				cm.state := 0;
//			END_IF

			pWorkStations.MC_BR_MoveInPlane_Acp6D_0.Shuttle := ADR(gAcp6DCtrl.Status.ShuttleInfo[pWorkStations.par.tempShuttleID].shuttleRef);
			pWorkStations.MC_BR_MoveInPlane_Acp6D_0.Parameters.Velocity := stainlessVelocity;
			pWorkStations.MC_BR_MoveInPlane_Acp6D_0.Parameters.Acceleration := stainlessAcceleration;
			pWorkStations.MC_BR_MoveInPlane_Acp6D_0.Parameters.Position.X := pWorkStations.par.xLocation;
			pWorkStations.MC_BR_MoveInPlane_Acp6D_0.Parameters.Position.Y := 0.060;

			pWorkStations.MC_BR_MoveInPlane_Acp6D_0.Execute := TRUE;
			IF pWorkStations.MC_BR_MoveInPlane_Acp6D_0.Done AND sheetMoveDone THEN
				pWorkStations.MC_BR_MoveInPlane_Acp6D_0.Execute := FALSE;
				cm.state := 35;
			END_IF

		35:
			pWorkStations.TON_0.IN := TRUE;
			pWorkStations.TON_0.PT := stainlessWaitTime;
			IF pWorkStations.TON_0.Q THEN
				pWorkStations.TON_0.IN := FALSE;
				cm.state := 10;
			END_IF

	END_CASE

	//Calls
	pWorkStations.MC_BR_MoveInPlane_Acp6D_0();
	pWorkStations.MC_BR_MoveArc_Acp6D_0();
	pWorkStations.MC_BR_Move6D_Acp6D_0();
	pWorkStations.MC_BR_ShLevitation_Acp6D_0();
	pWorkStations.MC_BR_RotaryMotion_Acp6D_0();
	pWorkStations.MC_BR_RotaryMotionSpin_Acp6D_0();
	pWorkStations.MC_BR_MoveShortAxis_Acp6D_0();
	pWorkStations.TON_0();
	cm();

END_ACTION
```

#### teachShuttle.st
```iecst
ACTION teachShuttleProgram:
	//setup
	positionContainerFlaskProgram[0].initXPos := 0.060;
	positionContainerFlaskProgram[0].initYPos := 0.060;
	positionContainerFlaskProgram[1].initXPos := 0.060;
	positionContainerFlaskProgram[1].initYPos := 0.180;
	positionContainerFlaskProgram[2].initXPos := 0.180;
	positionContainerFlaskProgram[2].initYPos := 0.120;
	positionContainerFlaskProgram[3].initXPos := 0.360;
	positionContainerFlaskProgram[3].initYPos := 0.120;
	CASE em.substate OF
		16000:
			em.cmd.sc := FALSE;
			em.description := 'Move shuttle to pre pos';
			tempShuttleCounter := 0;
			MC_BR_MoveInPlaneAsync_Acp6D_0.Parameters.Acceleration := gAcp6DCtrl.Par.Acceleration;
			MC_BR_MoveInPlaneAsync_Acp6D_0.Parameters.Velocity := gAcp6DCtrl.Par.Velocity;
			FOR i := 0 TO UINT_TO_USINT(localCurrentNumShuttles-1) DO
				MC_BR_MoveInPlaneAsync_Acp6D_0.Parameters.AsyncPar[i].Shuttle := ADR(gAcp6DCtrl.Status.ShuttleInfo[i].shuttleRef);
				MC_BR_MoveInPlaneAsync_Acp6D_0.Parameters.AsyncPar[i].X := positionContainerFlaskProgram[i].initXPos;
				MC_BR_MoveInPlaneAsync_Acp6D_0.Parameters.AsyncPar[i].Y := positionContainerFlaskProgram[i].initYPos;
			END_FOR
			MC_BR_MoveInPlaneAsync_Acp6D_0.Execute := TRUE;
			IF MC_BR_MoveInPlaneAsync_Acp6D_0.Done THEN
				MC_BR_MoveInPlaneAsync_Acp6D_0.Execute := FALSE;
				em.substate := 16010;
			END_IF

		16010:
			em.cmd.sc := FALSE;
			em.description := 'Deactivate segment 2';
			MC_BR_SegPowerOff_Acp6D_0.Segment := ADR(gAcp6DCtrl.Status.SegmentInfo[1].segmentRef);
			MC_BR_SegPowerOff_Acp6D_0.Execute := TRUE;
			IF MC_BR_SegPowerOff_Acp6D_0.Done THEN
				shuttleDeativatedLock := TRUE;
				MC_BR_SegPowerOff_Acp6D_0.Execute := FALSE;
				em.substate := 16020;
			END_IF

		16020:
			em.cmd.sc := FALSE;
			em.description := 'Menu';
			IF teachProgram.teachPosCmd THEN
				teachProgram.teachPosCmd := FALSE;
				em.substate := 16100;
			ELSIF teachProgram.runProgram THEN
				teachProgram.runProgram := FALSE;
				teachProgram.tmpRunPosCnt := 0;
				em.substate := 16200;
			ELSIF teachProgram.clearPositions THEN
				FOR i := 0 TO 99 DO
					teachProgram.positionArray[i].xPos := 0;
					teachProgram.positionArray[i].yPos := 0;
					teachProgram.savedPositions := 0;
				END_FOR
			ELSIF gAcp6DCtrl.Par.modeSelector <> teachProgramEnum THEN
				em.substate := 16300;
			END_IF

		16100:
			em.cmd.sc := FALSE;
			em.description := 'Teach Position';
			IF gAcp6DCtrl.Status.ShuttleInfo[3].State = mcACP6D_SH_STATE_DISABLED THEN
				teachProgram.positionArray[teachProgram.savedPositions].xPos := gAcp6DCtrl.Status.ShuttleInfo[3].Position.X;
				teachProgram.positionArray[teachProgram.savedPositions].yPos := gAcp6DCtrl.Status.ShuttleInfo[3].Position.Y;
//				teachProgram.positionArray[teachProgram.savedPositions].zPos := gAcp6DCtrl.Status.ShuttleInfo[3].Position.Z;
//				teachProgram.positionArray[teachProgram.savedPositions].rxPos := gAcp6DCtrl.Status.ShuttleInfo[3].Position.Rx;
//				teachProgram.positionArray[teachProgram.savedPositions].ryPos := gAcp6DCtrl.Status.ShuttleInfo[3].Position.Ry;
//				teachProgram.positionArray[teachProgram.savedPositions].rzPos := gAcp6DCtrl.Status.ShuttleInfo[3].Position.Rz;
				teachProgram.savedPositions := teachProgram.savedPositions + 1;
				em.substate := 16020;
			ELSE
				em.substate := 16020;
			END_IF

		16200:
			em.cmd.sc := FALSE;
			MC_BR_SegPowerOn_Acp6D_0.Segment := ADR(gAcp6DCtrl.Status.SegmentInfo[1].segmentRef);
			MC_BR_SegPowerOn_Acp6D_0.Execute := TRUE;
			IF MC_BR_SegPowerOn_Acp6D_0.Done THEN
				MC_BR_SegPowerOn_Acp6D_0.Execute := FALSE;
				em.substate := 16210;
			END_IF

		16210:
			em.cmd.sc := FALSE;
			em.description := 'Run teached program';
			IF teachProgram.tmpRunPosCnt >= teachProgram.savedPositions THEN
				em.substate := 16230;
			ELSE
				em.substate := 16220;
			END_IF

		16220:
			em.cmd.sc := FALSE;
			em.description := 'Run next position in program';
			MC_BR_Move6D_Acp6D_0.Shuttle := ADR(gAcp6DCtrl.Status.ShuttleInfo[3].shuttleRef);
			MC_BR_Move6D_Acp6D_0.Parameters.InPlane.Position.X := teachProgram.positionArray[teachProgram.tmpRunPosCnt].xPos;
			MC_BR_Move6D_Acp6D_0.Parameters.InPlane.Position.Y := teachProgram.positionArray[teachProgram.tmpRunPosCnt].yPos;
			MC_BR_Move6D_Acp6D_0.Parameters.ShortAxis.Position.Z := 0.001;
			MC_BR_Move6D_Acp6D_0.Parameters.InPlane.Velocity := gAcp6DCtrl.Par.Velocity;
			MC_BR_Move6D_Acp6D_0.Parameters.InPlane.Acceleration := gAcp6DCtrl.Par.Acceleration;
			MC_BR_Move6D_Acp6D_0.Parameters.ShortAxis.Velocity.Rx := 1;
			MC_BR_Move6D_Acp6D_0.Parameters.ShortAxis.Velocity.Ry := 1;
			MC_BR_Move6D_Acp6D_0.Parameters.ShortAxis.Velocity.Rz := 1;
			MC_BR_Move6D_Acp6D_0.Parameters.ShortAxis.Velocity.Z := 1;
			MC_BR_Move6D_Acp6D_0.Parameters.ShortAxis.Position.Rz := teachProgram.positionArray[teachProgram.tmpRunPosCnt].rzPos;
			MC_BR_Move6D_Acp6D_0.Execute := TRUE;
			IF MC_BR_Move6D_Acp6D_0.Done THEN
				MC_BR_Move6D_Acp6D_0.Execute := FALSE;
				teachProgram.tmpRunPosCnt := teachProgram.tmpRunPosCnt + 1;
				em.substate := 16210;
			END_IF

		16230:
			em.cmd.sc := FALSE;
			em.description := 'Turn off segment before reteaching';
			MC_BR_SegPowerOff_Acp6D_0.Segment := ADR(gAcp6DCtrl.Status.SegmentInfo[1].segmentRef);
			MC_BR_SegPowerOff_Acp6D_0.Execute := TRUE;
			IF MC_BR_SegPowerOff_Acp6D_0.Done THEN
				MC_BR_SegPowerOff_Acp6D_0.Execute := FALSE;
				em.substate := 16020;
			END_IF

		16300:
			em.cmd.sc := FALSE;
			em.description := 'Power on segment before program change';
			MC_BR_SegPowerOn_Acp6D_0.Segment := ADR(gAcp6DCtrl.Status.SegmentInfo[1].segmentRef);
			MC_BR_SegPowerOn_Acp6D_0.Execute := TRUE;
			IF MC_BR_SegPowerOn_Acp6D_0.Done THEN
				MC_BR_SegPowerOn_Acp6D_0.Execute := FALSE;
				em.substate := 16310;
			END_IF

		16310:
			em.description := 'Check that shuttle is rdy';
			IF gAcp6DCtrl.Status.ShuttleInfo[3].State = mcACP6D_SH_STATE_IDLING THEN
				MC_BR_SegBarrierCommand_Acp6D_0.Segment := ADR(gAcp6DCtrl.Status.SegmentInfo[1].segmentRef);
				MC_BR_SegBarrierCommand_Acp6D_0.Parameters.Command := mcACP6D_BARRIER_OPEN;
				MC_BR_SegBarrierCommand_Acp6D_0.Execute := TRUE;
				IF MC_BR_SegBarrierCommand_Acp6D_0.Done THEN
					MC_BR_SegBarrierCommand_Acp6D_0.Execute := FALSE;
					shuttleDeativatedLock := FALSE;
					em.cmd.sc := TRUE;
				END_IF
			END_IF

	END_CASE

END_ACTION
```

#### trakMode.st
```iecst
ACTION trakModeTask:

	CASE em.substate OF
		17000:
			em.cmd.sc := FALSE;
			em.description := 'Move shuttle to pre pos';
			positionContainerTrakMode[0].initXPos := 0.060;
			positionContainerTrakMode[0].initYPos := 0.060;
			positionContainerTrakMode[1].initXPos := 0.060;
			positionContainerTrakMode[1].initYPos := 0.180;
			positionContainerTrakMode[2].initXPos := 0.300;
			positionContainerTrakMode[2].initYPos := 0.180;
			positionContainerTrakMode[3].initXPos := 0.420;
			positionContainerTrakMode[3].initYPos := 0.180;
			tempShuttleCounter := 0;
			MC_BR_MoveInPlaneAsync_Acp6D_0.Parameters.Acceleration := gAcp6DCtrl.Par.Acceleration;
			MC_BR_MoveInPlaneAsync_Acp6D_0.Parameters.Velocity := gAcp6DCtrl.Par.Velocity;
			FOR i := 0 TO UINT_TO_USINT(localCurrentNumShuttles-1) DO
				MC_BR_MoveInPlaneAsync_Acp6D_0.Parameters.AsyncPar[i].Shuttle := ADR(gAcp6DCtrl.Status.ShuttleInfo[i].shuttleRef);
				MC_BR_MoveInPlaneAsync_Acp6D_0.Parameters.AsyncPar[i].X := positionContainerTrakMode[i].initXPos;
				MC_BR_MoveInPlaneAsync_Acp6D_0.Parameters.AsyncPar[i].Y := positionContainerTrakMode[i].initYPos;
			END_FOR
			MC_BR_MoveInPlaneAsync_Acp6D_0.Execute := TRUE;
			IF MC_BR_MoveInPlaneAsync_Acp6D_0.Done THEN
				MC_BR_MoveInPlaneAsync_Acp6D_0.Execute := FALSE;
				em.substate := 17010;
			END_IF

		17010:
		//HMI interface
			IF trakMode.bigBottle THEN
				em.substate := 17100;
				trakMode.bigBottle := FALSE;
			ELSIF trakMode.smallBottle THEN
				em.substate := 17200;
				trakMode.smallBottle := FALSE;
			END_IF

		17100:
			em.description := 'adjust shuttle to bigBottle';
			MC_BR_MoveInPlane_Acp6D_0.Shuttle := ADR(gAcp6DCtrl.Status.ShuttleInfo[2].shuttleRef);
			MC_BR_MoveInPlane_Acp6D_0.Parameters.Position.X := 0.276;
			MC_BR_MoveInPlane_Acp6D_0.Parameters.Position.Y := 0.180;
			MC_BR_MoveInPlane_Acp6D_0.Parameters.Velocity := gAcp6DCtrl.Par.Velocity;
			MC_BR_MoveInPlane_Acp6D_0.Parameters.Acceleration := gAcp6DCtrl.Par.Acceleration;
			MC_BR_MoveInPlane_Acp6D_0.Parameters.Mode := 0;
			MC_BR_MoveInPlane_Acp6D_0.Parameters.Path := 0;
			MC_BR_MoveInPlane_Acp6D_0.Execute := TRUE;
			IF MC_BR_MoveInPlane_Acp6D_0.Acknowledge THEN
				MC_BR_MoveInPlane_Acp6D_0.Execute := FALSE;
				em.substate := 17500;
			END_IF

		17200:
			em.description := 'adjust shuttle to smallBottle';
			MC_BR_MoveInPlane_Acp6D_0.Shuttle := ADR(gAcp6DCtrl.Status.ShuttleInfo[2].shuttleRef);
			MC_BR_MoveInPlane_Acp6D_0.Parameters.Position.X := 0.293;
			MC_BR_MoveInPlane_Acp6D_0.Parameters.Position.Y := 0.180;
			MC_BR_MoveInPlane_Acp6D_0.Parameters.Velocity := gAcp6DCtrl.Par.Velocity;
			MC_BR_MoveInPlane_Acp6D_0.Parameters.Acceleration := gAcp6DCtrl.Par.Acceleration;
			MC_BR_MoveInPlane_Acp6D_0.Parameters.Mode := 0;
			MC_BR_MoveInPlane_Acp6D_0.Parameters.Path := 0;
			MC_BR_MoveInPlane_Acp6D_0.Execute := TRUE;
			IF MC_BR_MoveInPlane_Acp6D_0.Acknowledge THEN
				MC_BR_MoveInPlane_Acp6D_0.Execute := FALSE;
				em.substate := 17500;
			END_IF

		17500:
			em.description := 'Couple ShuttleGroup3_4';
			em.cmd.sc := FALSE;
			MC_BR_ShGroupCoupleCtrl_Acp6D_0.ShuttleGroup := shGroupShuttle3_4;
			MC_BR_ShGroupCoupleCtrl_Acp6D_0.Parameters.Mode := 1;
			MC_BR_ShGroupCoupleCtrl_Acp6D_0.Parameters.Option := 1; //Couple
			MC_BR_ShGroupCoupleCtrl_Acp6D_0.Execute := TRUE;
			IF MC_BR_ShGroupCoupleCtrl_Acp6D_0.Done THEN
				MC_BR_ShGroupCoupleCtrl_Acp6D_0.Execute := FALSE;
				em.substate := 17550;
			END_IF

		17550:
			em.description := 'Wait timer';
			em.cmd.sc := FALSE;
			TON_0.PT := t#3s;
			TON_0.IN := TRUE;
			IF TON_0.Q THEN
				TON_0.IN := FALSE;
				em.substate := 17600;
			END_IF

		17600:
			em.description := 'Move bottle';
			em.cmd.sc := FALSE;
			MC_BR_MoveInPlane_Acp6D_0.Shuttle := ADR(gAcp6DCtrl.Status.ShuttleInfo[2].shuttleRef);
			MC_BR_MoveInPlane_Acp6D_0.Parameters.Position.X := 0.180;
			MC_BR_MoveInPlane_Acp6D_0.Parameters.Position.Y := 0.180;
			MC_BR_MoveInPlane_Acp6D_0.Parameters.Velocity := 0.5;
			MC_BR_MoveInPlane_Acp6D_0.Parameters.Acceleration := 0.5;
			MC_BR_MoveInPlane_Acp6D_0.Parameters.Mode := 0;
			MC_BR_MoveInPlane_Acp6D_0.Parameters.Path := 0;
			MC_BR_MoveInPlane_Acp6D_0.Execute := TRUE;
			IF MC_BR_MoveInPlane_Acp6D_0.Acknowledge THEN
				MC_BR_MoveInPlane_Acp6D_0.Execute := FALSE;
				em.substate := 17610;
			END_IF

		17610:
			em.description := 'Move bottle';
			em.cmd.sc := FALSE;
			MC_BR_MoveInPlane_Acp6D_0.Shuttle := ADR(gAcp6DCtrl.Status.ShuttleInfo[3].shuttleRef);
			MC_BR_MoveInPlane_Acp6D_0.Parameters.Position.X := 0.420;
			MC_BR_MoveInPlane_Acp6D_0.Parameters.Position.Y := 0.180;
			MC_BR_MoveInPlane_Acp6D_0.Parameters.Velocity := 0.5;
			MC_BR_MoveInPlane_Acp6D_0.Parameters.Acceleration := 0.5;
			MC_BR_MoveInPlane_Acp6D_0.Parameters.Mode := 0;
			MC_BR_MoveInPlane_Acp6D_0.Parameters.Path := 0;
			MC_BR_MoveInPlane_Acp6D_0.Execute := TRUE;
			IF MC_BR_MoveInPlane_Acp6D_0.Acknowledge THEN
				MC_BR_MoveInPlane_Acp6D_0.Execute := FALSE;
				em.substate := 17700;
			END_IF

		17700:
			em.description := 'DeCouple ShuttleGroup3_4';
			em.cmd.sc := FALSE;
			MC_BR_ShGroupCoupleCtrl_Acp6D_0.ShuttleGroup := shGroupShuttle3_4;
			MC_BR_ShGroupCoupleCtrl_Acp6D_0.Parameters.Option := 0; //DeCouple
			MC_BR_ShGroupCoupleCtrl_Acp6D_0.Execute := TRUE;
			IF MC_BR_ShGroupCoupleCtrl_Acp6D_0.Done THEN
				MC_BR_ShGroupCoupleCtrl_Acp6D_0.Execute := FALSE;
				em.substate := 17010;
			END_IF

	END_CASE

	TON_0();

END_ACTION
```

#### Types.typ - Local data types
```iecst
TYPE
	shuttle_typ : 	STRUCT
		cm : brdkCM;
		status : shuttle_status_typ;
		par : shuttle_par_typ;
		function : shuttle_function_typ;
	END_STRUCT;
	shuttle_status_typ : 	STRUCT
		dummy : USINT;
	END_STRUCT;
	shuttle_par_typ : 	STRUCT
		shuttleID : USINT;
	END_STRUCT;
	shuttle_function_typ : 	STRUCT
		MC_BR_Move6D_Acp6D_0 : MC_BR_Move6D_Acp6D;
		MC_BR_MoveShortAxis_Acp6D_0 : MC_BR_MoveShortAxis_Acp6D;
		MC_BR_ShGetPayload_Acp6D_0 : MC_BR_ShGetPayload_Acp6D;
		MC_BR_MoveInPlane_Acp6D_0 : MC_BR_MoveInPlane_Acp6D;
		TON_0 : TON;
	END_STRUCT;
	teachProgram_typ : 	STRUCT
		positionArray : ARRAY[0..99]OF shuttlePos;
		savedPositions : USINT;
		runProgram : BOOL;
		clearPositions : BOOL;
		teachPosCmd : BOOL;
		tmpRunPosCnt : USINT;
	END_STRUCT;
	shuttlePos : 	STRUCT
		xPos : REAL;
		yPos : REAL;
		zPos : REAL;
		rxPos : REAL;
		ryPos : REAL;
		rzPos : REAL;
	END_STRUCT;
	thisShuttleSetup : 	STRUCT
		Shuttle2 : shuttlePos;
		Shuttle3 : shuttlePos;
		Shuttle4 : shuttlePos;
		Shuttle1 : shuttlePos;
	END_STRUCT;
	gameMemory_typ : 	STRUCT
		shuttlesIDs : ARRAY[0..NUM_SHUTTLES]OF USINT;
		shuttlesLeft : USINT;
		shuttlesDead : ARRAY[0..NUM_SHUTTLES]OF BOOL;
		shuttlePicked : ARRAY[0..NUM_SHUTTLES]OF BOOL;
		startGame : BOOL;
		choosenRandomShuttle : UDINT;
		showHMIButton : BOOL;
		showStartBtnHMI : BOOL;
		playerNumeric : REAL;
		players : ARRAY[0..NUM_SHUTTLES]OF BOOL;
		loosingShuttlesIDs : ARRAY[0..NUM_SHUTTLES]OF USINT;
		winningShuttleID : USINT;
		showWinningNumber : BOOL;
	END_STRUCT;
	ABB_typ : 	STRUCT
		HomePositionReached : BOOL;
		startSmallWeightMovement : BOOL;
		returnBigWeightMovement : BOOL;
		returnSmallWeightMovement : BOOL;
		startBigWeightMovement : BOOL;
	END_STRUCT;
	trakMode_typ : 	STRUCT
		bigBottle : BOOL;
		smallBottle : BOOL;
	END_STRUCT;
END_TYPE
```

#### Variables.var - Local variables
```iecst
VAR
	NettimeLastCycle_us : DINT; (*Old nettime used to calculate Powerlink cycle time*)
	TON_Wait : TON;
	PowerlinkCycle_us : DINT;
	Wait : BOOL;
	TriggerTimeDelta_us : DINT; (*Delta time in microseconds to the next trigger*)
	TriggerPosDelta : LREAL; (*Delta position in units to the next trigger*)
	AxisPositionNow : LREAL;
	steelSheetFlyingHeight : REAL := 0.003;
	ABBRobot : ABB_typ;
	cm : REFERENCE TO brdkCM;
	ConveyorMovementWorkstation1Time : REAL := 1.5;
	ConveyorMovementWorkstation2Time : REAL := 4;
	createShGroup : USINT;
END_VAR
VAR RETAIN
	danfossWorkStation1NUMRotations : USINT := 5;
	danfossWorkStation1Timer : USINT := 8;
	danfossWorkStation2NUMRotations : USINT := 5;
	danfossWorkStation2Timer : USINT := 8;
END_VAR
VAR
	em : brdkEM;
	enableButtons : BOOL;
	fbPayload : REAL;
	flaskProgramAcceleration : REAL := 0.2;
	flaskProgramVelocity : REAL := 2;
	stainlessAcceleration : REAL := 1;
	stainlessVelocity : REAL := 0.2;
	stainlessWaitTime : TIME := T#250ms;
	levitationVelocity : REAL := 0.003;
	gameBrain : gameMemory_typ;
	gShuttles : ARRAY[0..NUM_SHUTTLES] OF shuttle_typ;
	i : USINT;
	j : USINT;
	k : USINT;
	localCurrentNumShuttles : UINT;
	MARGIN : REAL := 0.0059;
	macroCreater : USINT;
	oldNetTime : DINT;
	rotCnt : UDINT;
	deltaRad : REAL;
	correctedPosRz : REAL;
	skipRot : UDINT := 4;
	triggerPointRz : REAL := 1;
	maWindowLen : UINT := 5000;
	movingAverage : MTFilterMovingAverage;
	rzRad : REAL;
	rzSpeed : REAL;
	rzPosOld : REAL;
	MC_BR_RotaryMotion_Acp6D_0 : MC_BR_RotaryMotion_Acp6D;
	MC_BR_ShStop_Acp6D_0 : MC_BR_ShStop_Acp6D;
	MC_BR_AsmLevitation_Acp6D_0 : MC_BR_AsmLevitation_Acp6D;
	MC_BR_AsmGetInfo_Acp6D_0 : MC_BR_AsmGetInfo_Acp6D;
	MC_BR_MacroRun_Acp6D_0 : MC_BR_MacroRun_Acp6D;
	MC_BR_MacroSave_Acp6D_0 : MC_BR_MacroSave_Acp6D;
	MC_BR_SegBarrierCommand_Acp6D_0 : MC_BR_SegBarrierCommand_Acp6D;
	MC_BR_MacroCreate_Acp6D_0 : MC_BR_MacroCreate_Acp6D;
	MC_BR_AsmGetShuttle_Acp6D_0 : MC_BR_AsmGetShuttle_Acp6D;
	MC_BR_ReadCyclicPosition_Acp6D_1 : MC_BR_ReadCyclicPosition_Acp6D;
	MC_BR_ReadCyclicPosition_Acp6D_2 : MC_BR_ReadCyclicPosition_Acp6D;
	MC_BR_ReadCyclicPosition_Acp6D_3 : MC_BR_ReadCyclicPosition_Acp6D;
	MC_BR_ReadCyclicPosition_Acp6D_0 : MC_BR_ReadCyclicPosition_Acp6D;
	MC_BR_AsmPowerOff_Acp6D_0 : MC_BR_AsmPowerOff_Acp6D;
	MC_BR_AsmPowerOn_Acp6D_0 : MC_BR_AsmPowerOn_Acp6D;
	MC_BR_AsmReadStatus_Acp6D_0 : MC_BR_AsmReadStatus_Acp6D;
	MC_BR_AsmStop_Acp6D_0 : MC_BR_AsmStop_Acp6D;
	MC_BR_Move6D_Acp6D_0 : MC_BR_Move6D_Acp6D;
	MC_BR_MoveArc_Acp6D_0 : MC_BR_MoveArc_Acp6D;
	MC_BR_MoveInPlaneAsync_Acp6D_0 : MC_BR_MoveInPlaneAsync_Acp6D;
	MC_BR_MoveInPlane_Acp6D_0 : MC_BR_MoveInPlane_Acp6D;
	MC_BR_MoveShortAxis_Acp6D_0 : ARRAY[0..3] OF MC_BR_MoveShortAxis_Acp6D;
	MC_BR_MoveShortAxis_Acp6D_winner : MC_BR_MoveShortAxis_Acp6D;
	MC_BR_ShGroupAddShuttle_Acp6D_0 : MC_BR_ShGroupAddShuttle_Acp6D;
	MC_BR_ShGroupCoupleCtrl_Acp6D_0 : MC_BR_ShGroupCoupleCtrl_Acp6D;
	MC_BR_ShGroupCreate_Acp6D_0 : MC_BR_ShGroupCreate_Acp6D;
	MC_BR_ShGroupCreate_Acp6D_1 : MC_BR_ShGroupCreate_Acp6D;
	MC_BR_ShGroupCreate_Acp6D_2 : MC_BR_ShGroupCreate_Acp6D;
	MC_BR_ShGroupCreate_Acp6D_3 : MC_BR_ShGroupCreate_Acp6D;
	MC_BR_ShGroupGetInfo_Acp6D_0 : MC_BR_ShGroupGetInfo_Acp6D;
	MC_BR_ShLevitation_Acp6D_0 : MC_BR_ShLevitation_Acp6D;
	MC_BR_AsmGetSegment_Acp6D_0 : MC_BR_AsmGetSegment_Acp6D;
	MC_BR_SegPowerOn_Acp6D_0 : MC_BR_SegPowerOn_Acp6D;
	MC_BR_SegPowerOff_Acp6D_0 : MC_BR_SegPowerOff_Acp6D;
	MC_BR_RotaryMotionSpin_Acp6D_0 : MC_BR_RotaryMotionSpin_Acp6D;
	MC_BR_ShReadInfo_Acp6D_0 : ARRAY[0..NUM_SHUTTLES] OF MC_BR_ShReadInfo_Acp6D;
	MC_BR_AsmReset_Acp6D_0 : MC_BR_AsmReset_Acp6D;
	modeSelectorString : STRING[80];
	positionContainerTrakMode : ARRAY[0..3] OF shuttleStartup_typ;
	positionContainerBoxProgram : ARRAY[0..3] OF shuttleStartup_typ;
	positionContainerDemo_0 : ARRAY[0..3] OF shuttleStartup_typ;
	positionContainerDialGauge : ARRAY[0..3] OF shuttleStartup_typ;
	positionContainerFlaskProgram : ARRAY[0..3] OF shuttleStartup_typ;
	positionContainerGameProgram : ARRAY[0..3] OF shuttleStartup_typ;
	positionContainerLinkMovement : ARRAY[0..7] OF thisShuttleSetup;
	positionContainerLoosingShuttles : ARRAY[0..2] OF shuttleStartup_typ;
	positionContainerShuttleToConv : ARRAY[0..3] OF shuttleStartup_typ;
	positionContainerVisionMovement : ARRAY[0..3] OF shuttleStartup_typ;
	positionContainerWorkstationMov : ARRAY[0..3] OF shuttleStartup_typ;
	trakMode : trakMode_typ;
	positionDanfoss : ARRAY[0..3] OF shuttleStartup_typ;
	positionContainerSteelSheet : ARRAY[0..3] OF shuttleStartup_typ;
	positionContainerRotation : ARRAY[0..3] OF shuttleStartup_typ;
	posotionContainerSunMovement : ARRAY[0..3] OF shuttleStartup_typ;
	pShuttle : REFERENCE TO shuttle_typ;
	pWorkStations : REFERENCE TO workStation_typ;
	shGroupShuttle1_2 : UDINT;
	shGroupShuttle1_4 : UDINT;
	shGroupShuttle2_3 : UDINT;
	shGroupShuttle3_4 : UDINT;
	shuttle : USINT;
	shuttlePayload : REAL;
	shuttleToTakePictureOf : USINT;
	tempCounter : USINT;
	tempShuttleCnt : USINT;
	tempShuttleCounter : USINT;
	tempShuttleID : USINT;
	tmpCnt : USINT;
	TON_0 : TON;
	TON_watchdog : TON;
	visionFlipFlop : BOOL;
	visionLightTON : TON;
	watchPShuttle : {REDUND_UNREPLICABLE} USINT;
	watchPWorkstation : USINT;
	weightCalibration : REAL;
END_VAR
VAR RETAIN
	weightProgramFlyingHight : REAL := 1.48;
END_VAR
VAR
	WorkStation1MovementTimer : REAL := 1.5;
	teachProgram : teachProgram_typ;
	shuttleDeativatedLock : BOOL;
	WorkStation2And3MovementTimer : REAL := 4;
	deltaTimeUs : REAL;
	sheetMoveDone : BOOL;
	tempINT : INT;
	correctionValue : REAL;
END_VAR
```

### Types.typ
```iecst
TYPE
	gMain_par_typ : 	STRUCT
		itemsPrShuttle : INT;
		controlLight : BOOL;
	END_STRUCT;
	gMain_status_typ : 	STRUCT
		powerOff : INT;
		running : INT;
		powerOn : INT;
		itemsPrHour : INT;
		itemsPrMin : INT;
		error : INT;
	END_STRUCT;
	gMain_cmd_typ : 	STRUCT
		powerOff : BOOL;
		powerOn : BOOL;
		start : BOOL;
		pause : BOOL;
		reset : BOOL;
		stop : BOOL;
		restartCtrl : BOOL; (*WARNING: restarts 6D controller and PLC*)
		forceError : BOOL;
		resetStart : BOOL; (*Reset & start the program *)
		advanced : BOOL; (*Show advance options*)
		unlockPrgSelect : BOOL; (*Unlock the option to select different program*)
	END_STRUCT;
	gMain_typ : 	STRUCT
		par : gMain_par_typ;
		status : gMain_status_typ;
		cmd : gMain_cmd_typ;
	END_STRUCT;
END_TYPE
```

### Variables.var
```iecst
VAR
	gMain : gMain_typ;
	modeSelector : USINT;
END_VAR
VAR CONSTANT
	NUM_SHUTTLES : USINT := 3; (*4[0..3]*)
END_VAR
```

### Program Logical/Modules/Main/Main

#### Main.st
```iecst
PROGRAM _INIT
	em.setup.name := 'main';
	em();
	gMain.cmd.unlockPrgSelect := TRUE;

	MC_BR_AsmReboot_Acp6D_0.Assembly 		:= ADR(gAssembly6D_1);
	MC_BR_AsmHalt_Acp6D_0.Assembly			:= ADR(gAssembly6D_1);

END_PROGRAM

PROGRAM _CYCLIC

	IF gMain.cmd.forceError THEN
		em.cmd.abort := TRUE;
	END_IF

	IF gMain.cmd.restartCtrl THEN
		MC_BR_AsmReboot_Acp6D_0.Execute := TRUE;
		IF MC_BR_AsmReboot_Acp6D_0.Acknowledge OR MC_BR_AsmReboot_Acp6D_0.Error THEN
			SYSreset(TRUE, 1);
		END_IF
	END_IF

	// Statuslight
	gMain.status.powerOff := gMain.status.powerOn := gMain.status.running := gMain.status.error := 0;
	gAcp6DCtrl.Par.modeSelector := modeSelector;
	gAcp6DCtrl.Par.modeSelectorOld := modeSelectorOldValue;

	CASE em.state OF
		STATE_STOPPED:
			gMain.status.powerOff := 1;
			IF gMain.cmd.start THEN
				em.cmd.reset := TRUE;
				em.cmd.sc := TRUE;
			END_IF

		STATE_RESETTING:
			gMain.status.powerOn := 1;
			em.description := 'wait for sytem to reset variables';
			gMain.status.powerOn := 1;
			em.cmd.sc := TRUE;

		STATE_IDLE:
			gMain.status.powerOn := 1;
			em.description := 'wait for start cmd';
			TON_0.PT := t#500ms;
			TON_0.IN := TRUE;
			IF TON_0.Q THEN
				TON_0.IN := FALSE;
				em.cmd.sc := TRUE;
				em.cmd.start := TRUE;
			END_IF

		STATE_STARTING:
			gMain.status.powerOn := 1;
			em.description :='Wait for system to power on';
			em.cmd.sc := TRUE;

		STATE_EXECUTE:
			// New mode has been selected while old program is running.
			IF em.cmd.sc AND gAcp6DCtrl.Par.modeSelector <> modeSelectorOldValue THEN
				em.cmd.complete := TRUE;
			END_IF

			modeSelectorOldValue := gAcp6DCtrl.Par.modeSelector;
			gMain.status.running := 1;
			IF gMain.cmd.pause THEN
				gMain.cmd.pause := FALSE;
				em.cmd.hold := TRUE;
			END_IF

			IF gMain.cmd.stop THEN
				em.cmd.stop := TRUE;
			END_IF
			em.cmd.sc := TRUE;

		STATE_HOLDING:
			MC_BR_AsmHalt_Acp6D_0.Option := mcACP6D_HALT;
			MC_BR_AsmHalt_Acp6D_0.Execute := TRUE;
			IF MC_BR_AsmHalt_Acp6D_0.Done THEN
				MC_BR_AsmHalt_Acp6D_0.Execute := FALSE;
				em.cmd.sc := TRUE;
			END_IF

		STATE_HELD:
			IF gMain.cmd.start THEN
				em.cmd.sc		:= TRUE;
				em.cmd.start	:= TRUE;
			END_IF

		STATE_UNHOLDING:
			MC_BR_AsmHalt_Acp6D_0.Option := mcACP6D_CONTINUE;
			MC_BR_AsmHalt_Acp6D_0.Execute := TRUE;
			IF MC_BR_AsmHalt_Acp6D_0.Done THEN
				MC_BR_AsmHalt_Acp6D_0.Execute := FALSE;
				em.cmd.sc := TRUE;
			END_IF

		STATE_STOPPING:
			gMain.status.powerOff 								:= 1;
			em.cmd.sc											:= TRUE;

		STATE_ABORTED:
			gMain.status.error := 1;
			//gAcp6DCtrl.Cmd.PowerOff								:= TRUE;
			IF gMain.cmd.reset THEN
				em.cmd.clear									:= TRUE;
			END_IF
			em.cmd.sc											:= TRUE;

		STATE_CLEARING:
			em.cmd.sc := TRUE;

		STATE_COMPLETE:
			em.cmd.reset := TRUE;
			em.cmd.sc := TRUE;

		ELSE
			em.cmd.sc := TRUE;
	END_CASE

	(* Reset & start cmd *)
	IF EDGENEG(gMain.cmd.resetStart) THEN
		gMain.cmd.reset := FALSE;
		gMain.cmd.start := FALSE;
	ELSIF gMain.cmd.resetStart THEN
		gMain.cmd.reset := TRUE;
		gMain.cmd.start := TRUE;
	END_IF;

	em();
	TON_0();
	MC_BR_MoveInPlane_Acp6D_0();
	MC_BR_AsmHalt_Acp6D_0();
	MC_BR_AsmReboot_Acp6D_0();

END_PROGRAM

PROGRAM _EXIT
	(* Insert code here *)

END_PROGRAM
```

### Program Logical/RWS

#### Variables.var
```iecst
VAR
	BrAbbRwsCore_0 : BrAbbRwsCore;
	BrAbbRwsVariable_0 : BrAbbRwsVariable;
	xPos : REAL;
	state : INT;
	yPos : REAL;
	returnState : INT;
	TON_0 : TON;
	writeValue : BOOL;
	nWriteValue : REAL;
END_VAR
```

#### Main.st
```iecst
PROGRAM _INIT
	(* Insert code here *)
	BrAbbRwsCore_0.Enable := TRUE;
	BrAbbRwsCore_0.Parameters.UserName := 'Admin';
	BrAbbRwsCore_0.Parameters.Password := 'robotics';
	BrAbbRwsCore_0.Parameters.WebServerVersion := BR_ABB_RWS_VERSION_V2;
	BrAbbRwsCore_0.Parameters.HostPort := 443;
	BrAbbRwsCore_0.Parameters.Timeout := 0;
	BrAbbRwsCore_0.Parameters.SecureConfigName := 'mySSLConfig';

	IF DiagCpuIsSimulated() THEN
		BrAbbRwsCore_0.Parameters.ServerIP := '127.0.0.1';
	ELSE
		BrAbbRwsCore_0.Parameters.ServerIP := '192.168.125.1';
	END_IF;

END_PROGRAM

PROGRAM _CYCLIC
	(* Insert code here *)
	BrAbbRwsCore_0;

	IF NOT BrAbbRwsCore_0.Error THEN
		BrAbbRwsVariable_0.Ident := BrAbbRwsCore_0.Ident;
	END_IF;

	BrAbbRwsVariable_0.Parameters.Module := 'TeknologiaDemo25';
	BrAbbRwsVariable_0.Parameters.Task := 'T_ROB1';

	CASE state OF
		0:
			BrAbbRwsVariable_0.Enable := TRUE;
			TON_0.IN := TRUE;
			TON_0.PT := TIME#1s;
			TON_0;

			IF TON_0.Q THEN
				TON_0.IN := FALSE;
				TON_0;
				state := 1;
			END_IF;

		1:
			IF NOT BrAbbRwsVariable_0.Error THEN
				BrAbbRwsVariable_0.Parameters.Variable := 'bRobotPhaseDone';
				BrAbbRwsVariable_0.Value.DataAdress := ADR(gRobot.Status.phaseOK);
				BrAbbRwsVariable_0.Value.DataType := BR_ABB_RWS_VAR_BOOL;
				BrAbbRwsVariable_0.GetValue := TRUE;
				returnState := 2;
				state := 100;
			END_IF;

		2:
			IF NOT BrAbbRwsVariable_0.Error THEN
				BrAbbRwsVariable_0.Parameters.Variable := 'nRobotPhase';
				BrAbbRwsVariable_0.Value.DataAdress := ADR(gRobot.Status.phaseNum);
				BrAbbRwsVariable_0.Value.DataType := BR_ABB_RWS_VAR_NUM;
				BrAbbRwsVariable_0.GetValue := TRUE;
				returnState := 5;
				state := 100;
			END_IF;

		5:
			TON_0.IN := NOT (gRobot.liftCup OR gRobot.placeCup OR gRobot.moveRobotHome);
			TON_0.PT := TIME#500ms;
			TON_0;

			IF TON_0.Q THEN
				TON_0.IN := FALSE;
				TON_0;
				state := 1;
			ELSE
				IF gRobot.liftCup THEN
					BrAbbRwsVariable_0.Value.DataAdress := ADR(gRobot.CupCoordinate.X);
					BrAbbRwsVariable_0.Value.DataType := BR_ABB_RWS_VAR_NUM;
					BrAbbRwsVariable_0.Parameters.Variable := 'nPos_X';
					BrAbbRwsVariable_0.SetValue := TRUE;
					returnState := 6;
					state := 200;

				ELSIF gRobot.moveRobotHome THEN

					state := 7;
				ELSIF gRobot.placeCup THEN
					BrAbbRwsVariable_0.Value.DataAdress := ADR(gRobot.CupCoordinate.X);
					BrAbbRwsVariable_0.Value.DataType := BR_ABB_RWS_VAR_NUM;
					BrAbbRwsVariable_0.Parameters.Variable := 'nPos_X';
					BrAbbRwsVariable_0.SetValue := TRUE;
					returnState := 6;
					state := 200;
				ELSIF gRobot.AcoposWin THEN
					gRobot.AcoposWin := FALSE;
					writeValue := TRUE;
					BrAbbRwsVariable_0.Value.DataAdress := ADR(writeValue);
					BrAbbRwsVariable_0.Value.DataType := BR_ABB_RWS_VAR_BOOL;
					BrAbbRwsVariable_0.Parameters.Variable := 'bAcoposWin';
					BrAbbRwsVariable_0.SetValue := TRUE;
					returnState := 5;
					state := 200;
				END_IF;
			END_IF;

		6:
			BrAbbRwsVariable_0.Value.DataAdress := ADR(gRobot.CupCoordinate.Y);
			BrAbbRwsVariable_0.Value.DataType := BR_ABB_RWS_VAR_NUM;
			BrAbbRwsVariable_0.Parameters.Variable := 'nPos_Y';
			BrAbbRwsVariable_0.SetValue := TRUE;
			returnState := 7;
			state := 200;
		7:
			IF gRobot.liftCup THEN
				gRobot.liftCup := FALSE;
				BrAbbRwsVariable_0.Parameters.Variable := 'nAcoposCmd';
				nWriteValue := 2;
			ELSIF gRobot.placeCup THEN
				gRobot.placeCup := FALSE;
				BrAbbRwsVariable_0.Parameters.Variable := 'nAcoposCmd';
				nWriteValue := 3;
			ELSIF gRobot.moveRobotHome THEN
				gRobot.moveRobotHome := FALSE;
				BrAbbRwsVariable_0.Parameters.Variable := 'nAcoposCmd';
				nWriteValue := 1;
			END_IF;

			BrAbbRwsVariable_0.Value.DataAdress := ADR(nWriteValue);
			BrAbbRwsVariable_0.Value.DataType := BR_ABB_RWS_VAR_NUM;
			BrAbbRwsVariable_0.SetValue := TRUE;
			returnState := 5;
			state := 200;
		100:
			IF BrAbbRwsVariable_0.Done THEN
				BrAbbRwsVariable_0.GetValue := FALSE;
				state := returnState;
			END_IF;

		200:
			IF BrAbbRwsVariable_0.Done THEN
				writeValue := FALSE;
				BrAbbRwsVariable_0.SetValue := FALSE;
				state := returnState;
			END_IF;

	END_CASE;

	BrAbbRwsVariable_0;

END_PROGRAM

PROGRAM _EXIT
	(* Insert code here *)

END_PROGRAM
```

### Program Logical/test

#### Types.typ
```iecst
TYPE
	jpCoordinate : 	STRUCT
		x : REAL;
		y : REAL;
	END_STRUCT;
	jpLine : 	STRUCT
		a : REAL;
		b : REAL;
		c : REAL;
	END_STRUCT;
END_TYPE
```

#### Variables.var
```iecst
VAR
	shuttles : ARRAY[0..gMAX_INDEX_SHUTTLE] OF Acp6dShuttleType; (*Global shuttle list*)
	count : DINT;
	Y0 : REAL;
	X0 : REAL;
	Y1 : REAL;
	X1 : REAL;
	i : USINT;
	selection : ARRAY[0..gMAX_INDEX_SHUTTLE] OF brfiShuttleSelectionType;
END_VAR
(*Insert your comment here.*)
VAR
	point1 : jpCoordinate;
	point2 : jpCoordinate;
	point3 : jpCoordinate;
	line1 : jpLine;
	line2 : jpLine;
	slope : REAL;
END_VAR
```

#### Main.st
```iecst
PROGRAM _INIT
	(* Insert code here *)

	FOR i := 0 TO 7 DO
		shuttles[i].index := i;
		shuttles[i].position.value.X := 0.120 + (i MOD 4) * 0.120;
		IF i < 4 THEN
			shuttles[i].position.value.Y := 0.120;
		ELSE
			shuttles[i].position.value.Y := 0.240;
		END_IF;
	END_FOR;

END_PROGRAM

PROGRAM _CYCLIC
	(* Insert code here *)
	count := brfiShuttleSelect(ADR(shuttles), ADR(selection), X0, Y0, X1, Y1);

//	IF point1.x = point2.x THEN
//		slope := 0;
//	ELSE
//		slope := (point2.y-point1.y) / (point2.x - point1.x);
//	END_IF;
//
	line1.a := point2.y - point1.y;
	line1.b := point1.x - point2.x;
	line1.c := -(line1.a * point1.x + line1.b * point1.y);

	line2.a := point3.y - point2.y;
	line2.b := point2.x - point3.x;
	line2.c := -(line2.a * point2.x + line2.b * point2.y);

END_PROGRAM

PROGRAM _EXIT
	(* Insert code here *)

END_PROGRAM
```

Listed in the project but not available here: Logical/Libraries/brdkMU/brdkMU.typ, Logical/Libraries/brdkMU/brdkEM.typ, Logical/Libraries/brdkMU/brdkCM.typ, Logical/Libraries/brdkMU/brdkUM.typ, Logical/Libraries/brdkMU/brdkMU.var, Logical/Libraries/brdkMU/brdkMU.fun, Logical/Libraries/brdkMU/brdkEM.c, Logical/Libraries/brdkMU/brdkEMModeToA.c, Logical/Libraries/brdkMU/brdkEMStateToA.c, Logical/Libraries/brdkMU/brdkEMSleep.c, Logical/Libraries/brdkMU/brdkEM_func.h, Logical/Libraries/brdkMU/brdkEM_func.c, Logical/Libraries/brdkMU/brdkCM.c, Logical/Libraries/brdkMU/brdkCMChangeParent.c, Logical/Libraries/brdkMU/brdkCMSleep.c, Logical/Libraries/brdkMU/brdkCM_func.h, Logical/Libraries/brdkMU/brdkUM.c, Logical/Libraries/brdkMU/brdkUM_func.h, Logical/Libraries/brdkMU/brdkUM_func.c, Logical/Libraries/brdkMU/brdkMU_func.h, Logical/Libraries/brdkMU/brdkMU_func.c, Logical/Libraries/brdkSTR/brdkSTR.typ, Logical/Libraries/brdkSTR/brdkSTR.var, Logical/Libraries/brdkSTR/brdkSTR.fun, Logical/Libraries/brdkSTR/brdkStrAppendUdintToA.c, Logical/Libraries/brdkSTR/brdkStrAToDint.c, Logical/Libraries/brdkSTR/brdkStrAToUdint.c, Logical/Libraries/brdkSTR/brdkStrCat.c, Logical/Libraries/brdkSTR/brdkStrCatAtChar.c, Logical/Libraries/brdkSTR/brdkStrCharAt.c, Logical/Libraries/brdkSTR/brdkStrCharCount.c, Logical/Libraries/brdkSTR/brdkStrCmp.c, Logical/Libraries/brdkSTR/brdkStrCpy.c, Logical/Libraries/brdkSTR/brdkStrCrc32.c, Logical/Libraries/brdkSTR/brdkStrDintToA.c, Logical/Libraries/brdkSTR/brdkStrEncode.c, Logical/Libraries/brdkSTR/brdkStrFill.c, Logical/Libraries/brdkSTR/brdkStrFillUp.c, Logical/Libraries/brdkSTR/brdkStrIndexOf.c, Logical/Libraries/brdkSTR/brdkStrInsertAtPos.c, Logical/Libraries/brdkSTR/brdkStrIsAlphabet.c, Logical/Libraries/brdkSTR/brdkStrIsDigit.c, Logical/Libraries/brdkSTR/brdkStrIsEmpty.c, Logical/Libraries/brdkSTR/brdkStrJoin.c, Logical/Libraries/brdkSTR/brdkStrLen.c, Logical/Libraries/brdkSTR/brdkStrMemClear.c, Logical/Libraries/brdkSTR/brdkStrMemCmp.c, Logical/Libraries/brdkSTR/brdkStrMemCpy.c, Logical/Libraries/brdkSTR/brdkStrMemMove.c, Logical/Libraries/brdkSTR/brdkStrMemSet.c, Logical/Libraries/brdkSTR/brdkStrMove.c, Logical/Libraries/brdkSTR/brdkStrNCpy.c, Logical/Libraries/brdkSTR/brdkStrRemove.c, Logical/Libraries/brdkSTR/brdkStrRepeat.c, Logical/Libraries/brdkSTR/brdkStrReplace.c, Logical/Libraries/brdkSTR/brdkStrReverse.c, Logical/Libraries/brdkSTR/brdkStrReverseWords.c, Logical/Libraries/brdkSTR/brdkStrSearch.c, Logical/Libraries/brdkSTR/brdkStrSlice.c, Logical/Libraries/brdkSTR/brdkStrSplit.c, Logical/Libraries/brdkSTR/brdkStrSubDintSearch.c, Logical/Libraries/brdkSTR/brdkStrSubStr.c, Logical/Libraries/brdkSTR/brdkStrSubStrSearch.c, Logical/Libraries/brdkSTR/brdkStrToDec.c, Logical/Libraries/brdkSTR/brdkStrToHex.c, Logical/Libraries/brdkSTR/brdkStrToLowerCase.c, Logical/Libraries/brdkSTR/brdkStrToUpperCase.c, Logical/Libraries/brdkSTR/brdkStrToUpperCaseWords.c, Logical/Libraries/brdkSTR/brdkStrTrim.c, Logical/Libraries/brdkSTR/brdkStrUdintToA.c, Logical/Libraries/brdkSTR/brdkStrWord.c, Logical/Libraries/brdkSTR/brdkSTR_func.h, Logical/Libraries/brdkSTR/brdkSTR_func.c, Logical/Libraries/comUtil/utf8.c, Logical/Libraries/comUtil/utf8.h, Logical/Libraries/comUtil/sha1.c, Logical/Libraries/comUtil/sha1.h, Logical/Libraries/comUtil/base64.h, Logical/Libraries/comUtil/base64.c, Logical/Libraries/comUtil/parson.c, Logical/Libraries/comUtil/parson.h, Logical/Libraries/comUtil/rtkTypes.h, Logical/Libraries/comUtil/rtkTask.h, Logical/Libraries/comUtil/bootModeApi.h, Logical/Libraries/comUtil/arexport.h, Logical/Libraries/strUtil/parson.c, Logical/Libraries/strUtil/parson.h, Logical/Conf6D/parson.c, Logical/Conf6D/parson.h, Logical/Conf6D/rtkTypes.h, Logical/Conf6D/arexport.h, Logical/Modules/Acopos6D/Acopos6D/Danfoss.st, Logical/Modules/Acopos6D/Acopos6D/DemoProgram.st
